Fanuc KAREL source: CA0072.KL

-- PROVISIONAL review KL for V940-1; original PC SHA256 0cc3196aeceb714403542c74a9ad6d1181492d22d40bd7a0ddb8affe56f111ce
-- Incomplete behavior may be omitted. Consult companion uncertainty JSON. Do not deploy.
PROGRAM CA0072
%NOLOCKGROUP
BEGIN
  -- V9_ZERO_TABLE_METADATA_HINT layout=0001; no indexed target words; source/name/runtime held
  -- UNRESOLVED_PC offsets 0-1; opcodes 7B
  -- UNRESOLVED_PC offsets 6-20; opcodes 21,9D,52,23
  -- UNRESOLVED_PC offsets 25-29; opcodes 7F
  -- UNRESOLVED_PC offsets 34-41; opcodes 9C,23
  -- UNRESOLVED_PC offsets 46-53; opcodes 9D,23
  -- UNRESOLVED_PC offsets 58-69; opcodes 2E,23
  -- UNRESOLVED_PC offsets 74-81; opcodes 9D,23
  -- UNRESOLVED_PC offsets 86-95; opcodes 3F,75
  -- UNRESOLVED_PC offsets 100-114; opcodes 2E,22,9D,33,35
  -- UNRESOLVED_PC offsets 119-133; opcodes 2E,22,9D,33,35
  -- UNRESOLVED_PC offsets 138-153; opcodes 2E,22,32,35
  -- UNRESOLVED_PC offsets 158-173; opcodes 2E,22,32,35
  -- UNRESOLVED_PC offsets 178-404; opcodes 27,22,27,21,22,27,73,22,22,22,22,1C,22,27,21,22,27,21,22,2A,22,22,22,22,1C,22,22,27,21,22,27,73,22,22,22,22,1C,22,27,21,22,27,21,22,2A,22,AA
  -- UNRESOLVED_PC offsets 409-413; opcodes 7F
END CA0072
